INTERFACE List


METHOD Append : List
VAR_INPUT
	data	: ANY;
END_VAR
END_METHOD


PROPERTY Datatype : ListType
GET
END_GET
END_PROPERTY

PROPERTY DatatypeDefined : BOOL
GET
END_GET
END_PROPERTY


// Delete pointers
METHOD FB_exit : BOOL
VAR_INPUT
	bInCopyCode : BOOL; // if TRUE, the exit method is called for exiting an instance that is copied afterwards (online change).
END_VAR
END_METHOD


METHOD Get : BOOL
VAR_INPUT
	index		: INT; // Allow for indexing from end
	destination	: ANY;
END_VAR
END_METHOD


METHOD Insert : List
VAR_INPUT
	index	: INT; // Allow for indexing from end
	data	: ANY;
END_VAR
END_METHOD


METHOD IsEmpty : BOOL
VAR_INPUT
END_VAR
END_METHOD


METHOD IsTypeCorrect : BOOL
VAR_INPUT
	checkedVariable		: ANY;
END_VAR
END_METHOD


PROPERTY LastIndex : ListLength
GET
END_GET
END_PROPERTY


PROPERTY Length : ListLength
GET
END_GET
END_PROPERTY


METHOD Prepend : List
VAR_INPUT
	data	: ANY;
END_VAR
END_METHOD


METHOD Remove : List
VAR_INPUT
	index	: INT; // Allow for indexing from end
END_VAR
END_METHOD


METHOD RemoveAll : List
VAR_INPUT
END_VAR
END_METHOD


METHOD Set : List
VAR_INPUT
	index	: INT; // Allow for indexing from end
	data	: ANY;
END_VAR
END_METHOD

END_INTERFACE

(* stored: Version 1.1.0.1, ProductVersion 3.1.4024.12
   Itf List: Id {70fa5247-5b57-4846-9db9-81ed1f26b16a}
   Method Append: Id {a92455fb-c069-4c4d-8706-764afa701dba}
   Property Datatype: Id {c6bc2699-1bee-49b5-be56-8ebb92af4cdf}
   Get Get: Id {b138e580-5c0c-42fd-b580-7eb9da2885e9}
   Property DatatypeDefined: Id {9d9d2533-09e2-48b3-929a-fc5d087ac217}
   Get Get: Id {8ddb38aa-4597-45c4-ad8a-1daaa68377b4}
   Method FB_exit: Id {6a8bb466-a584-4df4-a32c-5c0774398859}
   Method Get: Id {824eaf5e-6f8d-432d-b9b2-1ece3ecf030d}
   Method Insert: Id {4d53e841-01dc-4246-9b49-a63507f8c33f}
   Method IsEmpty: Id {6803efab-caed-4135-a376-bebd90afd91b}
   Method IsTypeCorrect: Id {b8da7858-f130-4783-a1e0-771bc653b1c9}
   Property LastIndex: Id {e3810565-2d19-431d-b7d8-71f6d7ac8445}
   Get Get: Id {33f96068-472a-4358-9760-71610ab326e1}
   Property Length: Id {75637133-746b-4a7a-a424-c47794c6c5a7}
   Get Get: Id {f28c7547-3df9-456c-8f29-f927ce37b999}
   Method Prepend: Id {7546d95c-bb34-4096-8df9-689a87c4271c}
   Method Remove: Id {ef067663-f6a4-4c4f-a4f7-a2422263ba02}
   Method RemoveAll: Id {52c369d5-946b-41da-9dcf-b0be62710028}
   Method Set: Id {6c6bbffc-6a30-40ea-994d-315294a55206} *)
